KUKA KRL data list: vw_usr_s.dat

&ACCESS RV
&PARAM TPVW_VERSION = 3.3.5
DEFDAT  VW_USR_S
; FOLD ;%{H}%MKUKATPVW
; ENDFOLD
ENDDAT
